// TIA Portal V15.1 export
// export: Created 2024-05-17T05:38:13.3663523Z, ExportSetting WithDefaults, DisplayName Totally Integrated Automation Portal, DisplayVersion V15.1 Update 5, DisplayName TIA Portal Openness, DisplayVersion V15.1 Update 5, DisplayName SINAMICS Startdrive Advanced, DisplayVersion V15.1, DisplayName G130, G150, S120, S150, SINAMICS MV, S210, DisplayVersion V15.1, DisplayName G110M, G120, G120C, G120D, G120P, DisplayVersion V15.1, DisplayName STEP 7 Professional, DisplayVersion V15.1 Update 5, DisplayName STEP 7 Safety, DisplayVersion V15.1, DisplayName WinCC Professional, DisplayVersion V15.1 Update 5, DisplayName SIMATIC Visualization Architect, DisplayVersion V15.1
DATA_BLOCK "_209000NCP01EnableAlarms"   // DB198
{ S7_Optimized_Access := 'FALSE' }
VERSION : 0.1
// stored: AutoNumber false, DBAccessibleFromOPCUA true, IsOnlyStoredInLoadMemory false, IsWriteProtectedInAS false
   VAR RETAIN
      "General24VDC_AE01-AE02" { ExternalAccessible := 'False'; ExternalVisible := 'False'; ExternalWritable := 'False'} : Bool;   // General 24VDC - AE01 ... AE02
      "General24VDC_AK01-AK04" { ExternalAccessible := 'False'; ExternalVisible := 'False'; ExternalWritable := 'False'} : Bool;   // General 24VDC - AK01 ... AK04
      "209000AE02-JW210" { ExternalAccessible := 'False'; ExternalVisible := 'False'; ExternalWritable := 'False'} : Bool;   // General Switch - JW210
      "209210Field-JW221" { ExternalAccessible := 'False'; ExternalVisible := 'False'; ExternalWritable := 'False'} : Bool;   // Field Switch - JW221
      "209220Field-JW222" { ExternalAccessible := 'False'; ExternalVisible := 'False'; ExternalWritable := 'False'} : Bool;   // Field Switch - JW222
      "209230Field-JW223" { ExternalAccessible := 'False'; ExternalVisible := 'False'; ExternalWritable := 'False'} : Bool;   // Field Switch - JW223
      "209000AE01_24VDCFuse" { ExternalAccessible := 'False'; ExternalVisible := 'False'; ExternalWritable := 'False'} : Bool;   // 24VDC Fuses AE01
      "209000AK02_24VDCFuse" { ExternalAccessible := 'False'; ExternalVisible := 'False'; ExternalWritable := 'False'} : Bool;   // 24VDC Fuses AK02
      "209000AK01-JW35_IO" { ExternalAccessible := 'False'; ExternalVisible := 'False'; ExternalWritable := 'False'} : Bool;   // Busnode 000AK01 Input - Output
      "209000AK01-JW35_SafetyIO" { ExternalAccessible := 'False'; ExternalVisible := 'False'; ExternalWritable := 'False'} : Bool;   // Busnode 000AK01 Safety Input - Output
      "209000AK03-JW36_IO" { ExternalAccessible := 'False'; ExternalVisible := 'False'; ExternalWritable := 'False'} : Bool;   // Busnode 000AK03 Input - Output
      "209000AK03-JW36_SafetyIO" { ExternalAccessible := 'False'; ExternalVisible := 'False'; ExternalWritable := 'False'} : Bool;   // Busnode 000AK03 Safety Input - Output
      "209000AK04-JW37_IO" { ExternalAccessible := 'False'; ExternalVisible := 'False'; ExternalWritable := 'False'} : Bool;   // Busnode 000AK04 Input - Output
      "209000AK04-JW37_SafetyIO" { ExternalAccessible := 'False'; ExternalVisible := 'False'; ExternalWritable := 'False'} : Bool;   // Busnode 000AK04 Safety Input - Output
      "209000AS01-JW38_IO" { ExternalAccessible := 'False'; ExternalVisible := 'False'; ExternalWritable := 'False'} : Bool;   // Busnode 000AS01 Input - Output
      "209000AS01-JW38_SafetyIO" { ExternalAccessible := 'False'; ExternalVisible := 'False'; ExternalWritable := 'False'} : Bool;   // Busnode 000AS01 Safety Input - Output
      "209000AS02-JW39_IO" { ExternalAccessible := 'False'; ExternalVisible := 'False'; ExternalWritable := 'False'} : Bool;   // Busnode 000AS02 Input - Output
      "209000AS02-JW39_SafetyIO" { ExternalAccessible := 'False'; ExternalVisible := 'False'; ExternalWritable := 'False'} : Bool;   // Busnode 000AS02 Safety Input - Output
      "209210AS10-JW40_IO" { ExternalAccessible := 'False'; ExternalVisible := 'False'; ExternalWritable := 'False'} : Bool;   // Busnode 210AS10 Input - Output
      "209210AS10-JW40_SafetyIO" { ExternalAccessible := 'False'; ExternalVisible := 'False'; ExternalWritable := 'False'} : Bool;   // Busnode 210AS10 Safety Input - Output
      "209210AX01-JW41_IO" { ExternalAccessible := 'False'; ExternalVisible := 'False'; ExternalWritable := 'False'} : Bool;   // Busnode 210AX01 Input - Output
      "209210AX01-JW41_SafetyIO" { ExternalAccessible := 'False'; ExternalVisible := 'False'; ExternalWritable := 'False'} : Bool;   // Busnode 210AX01 Safety Input - Output
      "209210AS11-JW42_IO" { ExternalAccessible := 'False'; ExternalVisible := 'False'; ExternalWritable := 'False'} : Bool;   // Busnode 210AS11 Input - Output
      "209210AS11-JW42_SafetyIO" { ExternalAccessible := 'False'; ExternalVisible := 'False'; ExternalWritable := 'False'} : Bool;   // Busnode 210AS11 Safety Input - Output
      "209210AX02-JW43_IO" { ExternalAccessible := 'False'; ExternalVisible := 'False'; ExternalWritable := 'False'} : Bool;   // Busnode 210AX02 Input - Output
      "209210AX02-JW43_SafetyIO" { ExternalAccessible := 'False'; ExternalVisible := 'False'; ExternalWritable := 'False'} : Bool;   // Busnode 210AX02 Safety Input - Output
      "209210AS20-JW48_IO" { ExternalAccessible := 'False'; ExternalVisible := 'False'; ExternalWritable := 'False'} : Bool;   // Busnode 210AS20 Input - Output
      "209210AS20-JW48_SafetyIO" { ExternalAccessible := 'False'; ExternalVisible := 'False'; ExternalWritable := 'False'} : Bool;   // Busnode 210AS20 Safety Input - Output
      "209220AS10-JW50_IO" { ExternalAccessible := 'False'; ExternalVisible := 'False'; ExternalWritable := 'False'} : Bool;   // Busnode 220AS10 Input - Output
      "209220AS10-JW50_SafetyIO" { ExternalAccessible := 'False'; ExternalVisible := 'False'; ExternalWritable := 'False'} : Bool;   // Busnode 220AS10 Safety Input - Output
      "209220AX01-JW51_IO" { ExternalAccessible := 'False'; ExternalVisible := 'False'; ExternalWritable := 'False'} : Bool;   // Busnode 220AX01 Input - Output
      "209220AX01-JW51_SafetyIO" { ExternalAccessible := 'False'; ExternalVisible := 'False'; ExternalWritable := 'False'} : Bool;   // Busnode 220AX01 Safety Input - Output
      "209220AS11-JW52_IO" { ExternalAccessible := 'False'; ExternalVisible := 'False'; ExternalWritable := 'False'} : Bool;   // Busnode 220AS11 Input - Output
      "209220AS11-JW52_SafetyIO" { ExternalAccessible := 'False'; ExternalVisible := 'False'; ExternalWritable := 'False'} : Bool;   // Busnode 220AS11 Safety Input - Output
      "209220AX02-JW53_IO" { ExternalAccessible := 'False'; ExternalVisible := 'False'; ExternalWritable := 'False'} : Bool;   // Busnode 220AX02 Input - Output
      "209220AX02-JW53_SafetyIO" { ExternalAccessible := 'False'; ExternalVisible := 'False'; ExternalWritable := 'False'} : Bool;   // Busnode 220AX02 Safety Input - Output
      "209220AS20-JW58_IO" { ExternalAccessible := 'False'; ExternalVisible := 'False'; ExternalWritable := 'False'} : Bool;   // Busnode 220AS20 Input - Output
      "209220AS20-JW58_SafetyIO" { ExternalAccessible := 'False'; ExternalVisible := 'False'; ExternalWritable := 'False'} : Bool;   // Busnode 220AS20 Safety Input - Output
      "209230AS10-JW60_IO" { ExternalAccessible := 'False'; ExternalVisible := 'False'; ExternalWritable := 'False'} : Bool;   // Busnode 230AS10 Input - Output
      "209230AS10-JW60_SafetyIO" { ExternalAccessible := 'False'; ExternalVisible := 'False'; ExternalWritable := 'False'} : Bool;   // Busnode 230AS10 Safety Input - Output
      "209230AX01-JW61_IO" { ExternalAccessible := 'False'; ExternalVisible := 'False'; ExternalWritable := 'False'} : Bool;   // Busnode 230AX01 Input - Output
      "209230AX01-JW61_SafetyIO" { ExternalAccessible := 'False'; ExternalVisible := 'False'; ExternalWritable := 'False'} : Bool;   // Busnode 230AX01 Safety Input - Output
      "209210DriveMoviDrive" { ExternalAccessible := 'False'; ExternalVisible := 'False'; ExternalWritable := 'False'} : Bool;   // Drive 210 MoviDrive
      "209210DriveMoviFit" { ExternalAccessible := 'False'; ExternalVisible := 'False'; ExternalWritable := 'False'} : Bool;   // Drive 210 MoviFit
      "209220DriveMoviDrive" { ExternalAccessible := 'False'; ExternalVisible := 'False'; ExternalWritable := 'False'} : Bool;   // Drive 220 MoviDrive
      "209220DriveMoviFit" { ExternalAccessible := 'False'; ExternalVisible := 'False'; ExternalWritable := 'False'} : Bool;   // Drive 220 MoviFit
      "209230DriveMoviFit" { ExternalAccessible := 'False'; ExternalVisible := 'False'; ExternalWritable := 'False'} : Bool;   // Drive 230 MoviFit
      "209230MGB" { ExternalAccessible := 'False'; ExternalVisible := 'False'; ExternalWritable := 'False'} : Bool;   // Euchner Door 230
   END_VAR
BEGIN
END_DATA_BLOCK
